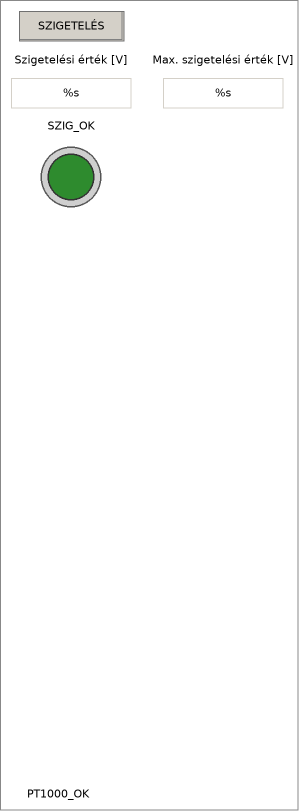
VISUALIZATION Vegmero_szigeteles  // 299x811
    Lamp1 (36,142 70x70), variable: NOT VEGMERO.bISOL_OK, style: Lamp-Lamp1-Red
    Label (36,116 70x20), "SZIG_OK"
    Button (19,11 105x30), "SZIGETELÉS", input disabled if: VEGMERO.s_InCommand<>''
        OnMouseUp: execute { VEGMERO.s_InCommand:='ATUTES'; }
    Textfield (11,78 120x30), "%s", text variable: VEGMERO.rISOL
    Label (11,50 120x20), "Szigetelési érték [V]"
    Label (3,779 110x30), "PT1000_OK"
    Textfield (163,78 120x30), "%s", text variable: GVL.rISOL_MAX
    Label (149,50 148x20), "Max. szigetelési érték [V]"
    Lamp1 (36,142 70x70), variable: VEGMERO.bISOL_OK, invisible if: NOT VEGMERO.bISOL_OK AND VEGMERO.bISOL_MERVE, style: Lamp-Lamp1-Green
END_VISUALIZATION

(* stored: Version 1.1.0.1, ProductVersion 3.1.4024.11
   Visu Vegmero_szigeteles: Id {c81eef93-3e1c-4e25-9774-9df4045be223} *)
